// Mitsubishi GX Works2 project: PART_B_ready_with light   PLC: FX3G

// global labels: Global1
VAR_GLOBAL
  new_order AT X007 : BOOL;
  REG_orders AT D1112 : REAL;
END_VAR
VAR_GLOBAL CONSTANT
  const1 : REAL := 1;
END_VAR
VAR_GLOBAL
  PanWeightSen AT X003 : BOOL;
  work_day AT X000 : BOOL;
END_VAR
VAR_GLOBAL CONSTANT
  twoMin : INT := 1200;
  tenSec : INT := 100;
END_VAR
VAR_GLOBAL
  TC_cookingTimer AT TC0 : BOOL;
  TCFI_fifteen_noodels AT TC2 : BOOL;
END_VAR
VAR_GLOBAL CONSTANT
  const15 : INT := 150;
END_VAR
VAR_GLOBAL
  dishReady AT M111 : BOOL;
END_VAR
VAR_GLOBAL CONSTANT
  const_fifteen : INT := 150;
END_VAR
VAR_GLOBAL
  is_VEG_COOKED AT TS0 : BOOL;
  IS_dish_cooked AT TS2 : BOOL;
  iscooked AT M1 : BOOL;
  dayInProcess AT Y000 : BOOL;
  REG_waiting_orders AT D1114 : REAL;
  startCooking AT M1 : BOOL;
  new_order_added AT M3 : BOOL;
END_VAR
VAR_GLOBAL CONSTANT
  const0 : REAL;
END_VAR
VAR_GLOBAL
  REG_done AT D1117 : REAL;
  Pulse AT X002 : BOOL;
  sen100 AT X004 : BOOL;
  sen90 AT X005 : BOOL;
  heatPan AT M135 : BOOL;
  veg_inventory AT D1119 : REAL;
END_VAR
VAR_GLOBAL CONSTANT
  GRAM100 : REAL := 100;
END_VAR
VAR_GLOBAL
  REG_pan_weight AT D4000 : REAL;
  enough_Veg_On_Pan AT M14 : BOOL;
  noodles_inventory AT D1202 : REAL;
  enough_noodles_on_pan AT M16 : BOOL;
END_VAR
VAR_GLOBAL CONSTANT
  kg3 : REAL := 3000;
  GRAM200 : REAL := 200;
END_VAR
VAR_GLOBAL
  Pan_is_hot AT M44 : BOOL;
  hot_pan_needed AT M13 : BOOL;
  order_is_up AT M12 : BOOL;
  is_served AT M32 : BOOL;
END_VAR

// task Task_01 (event TRUE, interval 0, priority 31): POU_01

PROGRAM POU_01
(* structured ladder/FBD written out as ST: instructions are called as NAME(EN, inputs, outputs); _pN, _eN, _tN stand for wires *)
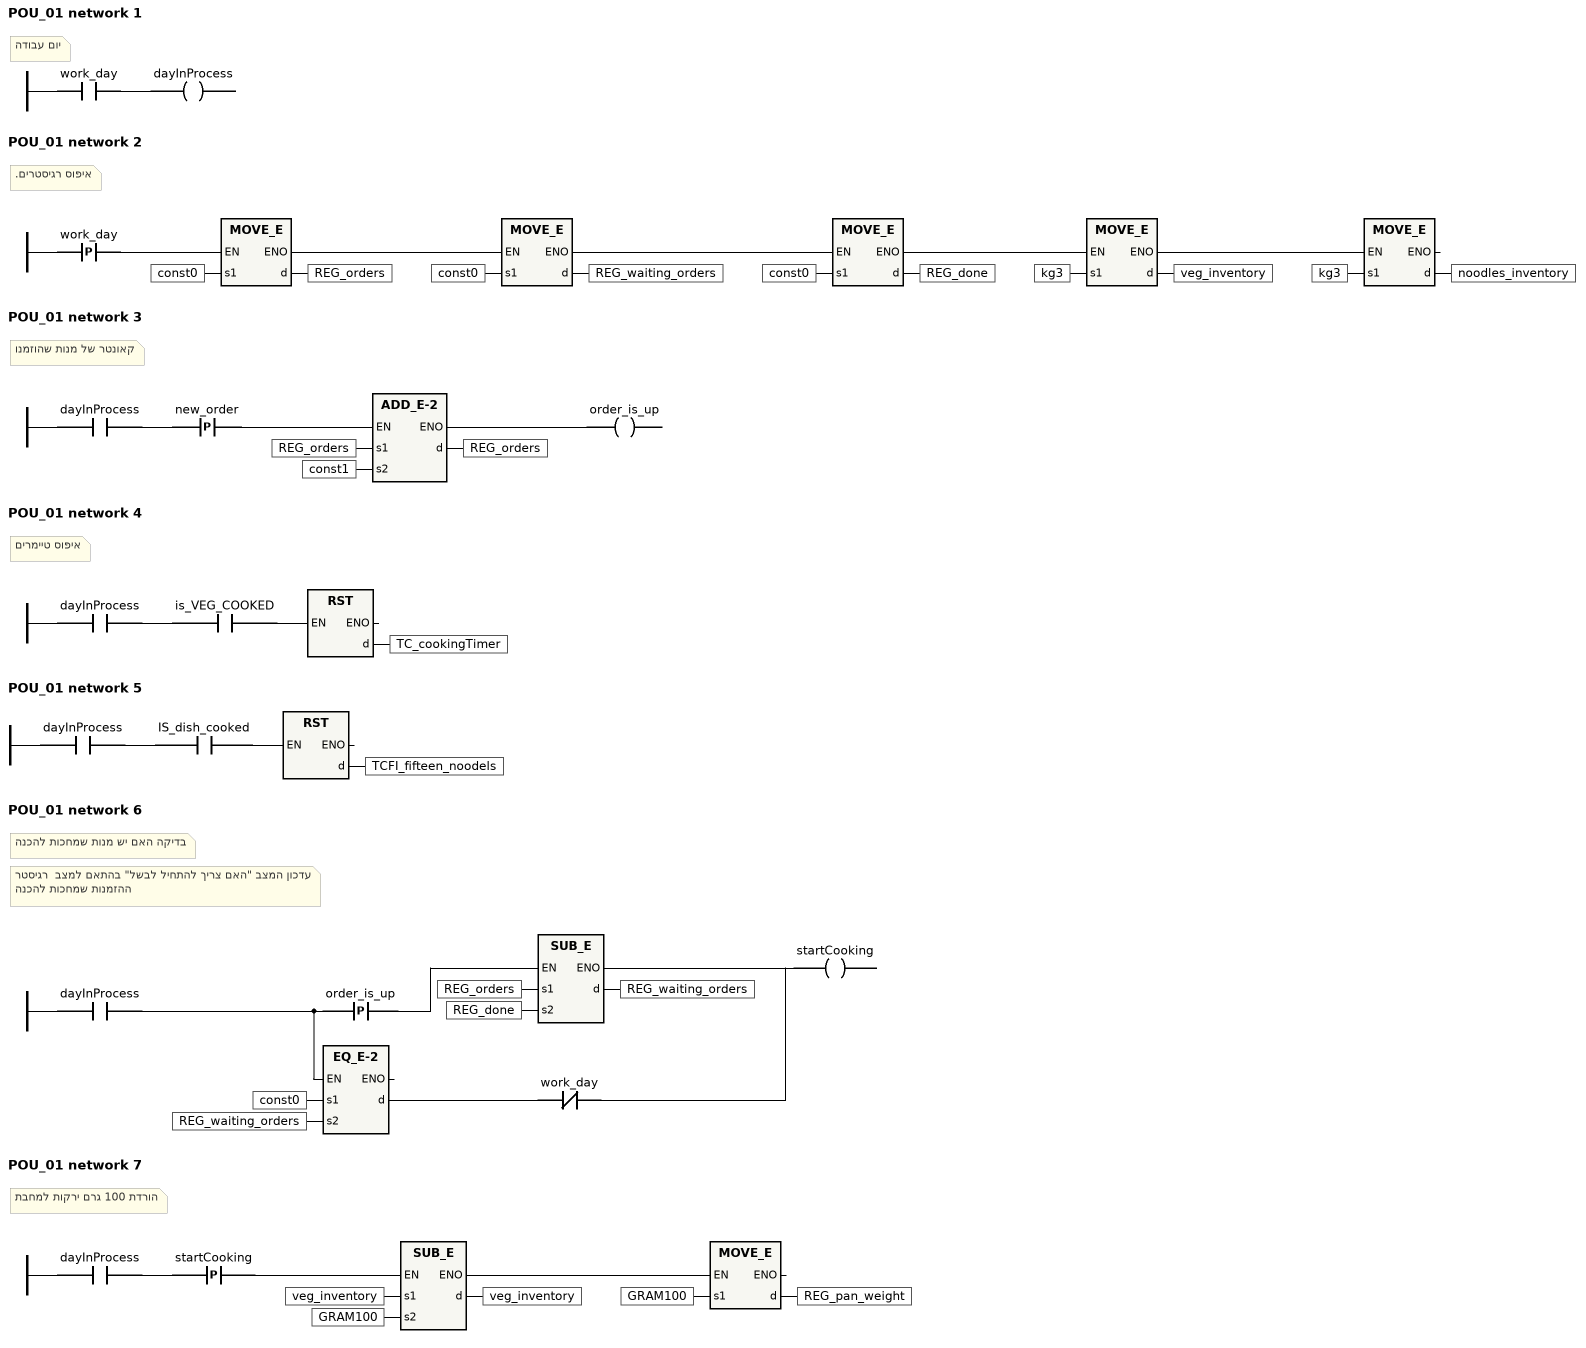
(* network 1 1 *)
(* יום עבודה *)
dayInProcess := work_day;
(* network 2 *)
(* איפוס רגיסטרים. *)
_e1 := MOVE_E(LDP(TRUE, work_day), const0, REG_orders);
_e2 := MOVE_E(_e1, const0, REG_waiting_orders);
_e3 := MOVE_E(_e2, const0, REG_done);
_e4 := MOVE_E(_e3, kg3, veg_inventory);
MOVE_E(_e4, kg3, noodles_inventory);
(* network 3 *)
(* קאונטר של מנות שהוזמנו *)
_e1 := ADD_E(dayInProcess AND LDP(TRUE, new_order), REG_orders, const1, REG_orders);
order_is_up := _e1;
(* network 4 *)
(* איפוס טיימרים *)
RST(dayInProcess AND is_VEG_COOKED, TC_cookingTimer);
(* network 5 *)
RST(dayInProcess AND IS_dish_cooked, TCFI_fifteen_noodels);
(* network 6 *)
(* בדיקה האם יש מנות שמחכות להכנה *)
(* עדכון המצב "האם צריך להתחיל לבשל" בהתאם למצב  רגיסטר ההזמנות שמחכות להכנה *)
_e1 := SUB_E(dayInProcess AND LDP(TRUE, order_is_up), REG_orders, REG_done, REG_waiting_orders);
EQ_E(dayInProcess, const0, REG_waiting_orders, _t2);
startCooking := _e1 OR (_t2 AND NOT work_day);
(* network 7 *)
(* הורדת 100 גרם ירקות למחבת *)
_e1 := SUB_E(dayInProcess AND LDP(TRUE, startCooking), veg_inventory, GRAM100, veg_inventory);
MOVE_E(_e1, GRAM100, REG_pan_weight);
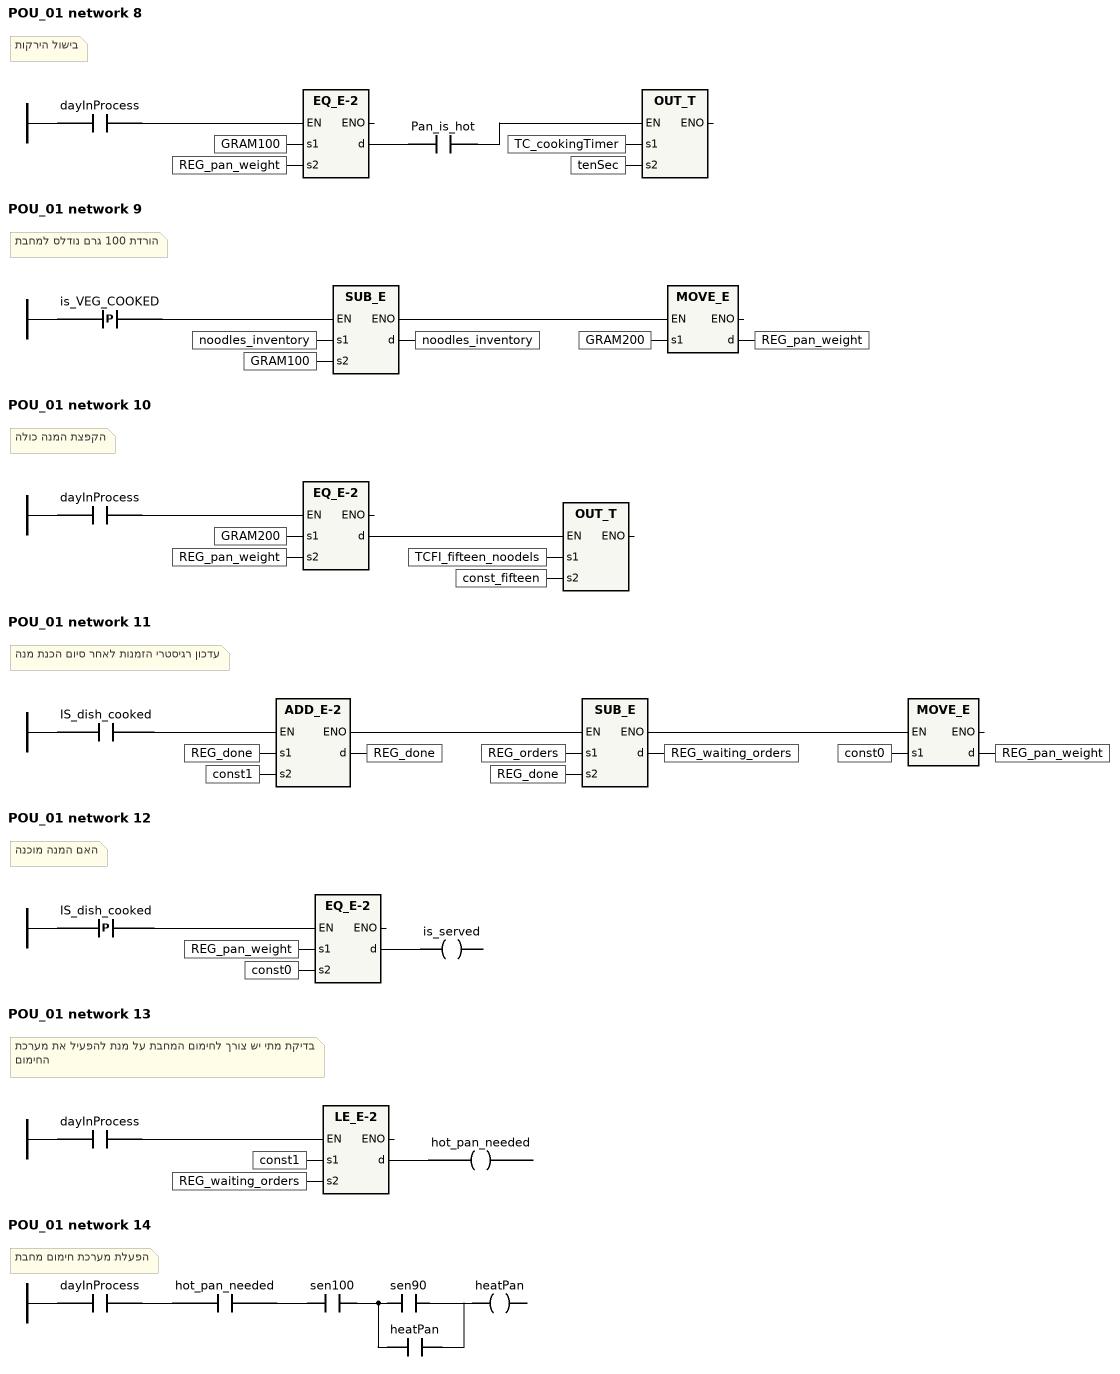
(* network 8 *)
(* בישול הירקות *)
EQ_E(dayInProcess, GRAM100, REG_pan_weight, _t1);
OUT_T(_t1 AND Pan_is_hot, TC_cookingTimer, tenSec);
(* network 9 *)
(* הורדת 100 גרם נודלס למחבת *)
_e1 := SUB_E(LDP(TRUE, is_VEG_COOKED), noodles_inventory, GRAM100, noodles_inventory);
MOVE_E(_e1, GRAM200, REG_pan_weight);
(* network 10 *)
(* הקפצת המנה כולה *)
EQ_E(dayInProcess, GRAM200, REG_pan_weight, _t1);
OUT_T(_t1, TCFI_fifteen_noodels, const_fifteen);
(* network 11 *)
(* עדכון רגיסטרי הזמנות לאחר סיום הכנת מנה *)
_e1 := ADD_E(IS_dish_cooked, REG_done, const1, REG_done);
_e2 := SUB_E(_e1, REG_orders, REG_done, REG_waiting_orders);
MOVE_E(_e2, const0, REG_pan_weight);
(* network 12 *)
(* האם המנה מוכנה *)
EQ_E(LDP(TRUE, IS_dish_cooked), REG_pan_weight, const0, _t1);
is_served := _t1;
(* network 13 *)
(* בדיקת מתי יש צורך לחימום המחבת על מנת להפעיל את מערכת החימום *)
LE_E(dayInProcess, const1, REG_waiting_orders, _t1);
hot_pan_needed := _t1;
(* network 14 *)
(* הפעלת מערכת חימום מחבת *)
_p1 := dayInProcess AND hot_pan_needed AND sen100;
heatPan := (_p1 AND sen90) OR (_p1 AND heatPan);
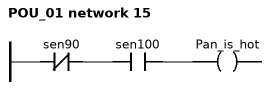
(* network 15 *)
Pan_is_hot := NOT sen90 AND sen100;
END_PROGRAM
